FUNCTION_BLOCK FB_Alarm EXTENDS Tc3_EventLogger.FB_TcAlarm
VAR_INPUT
	stEventEntry : TcEventEntry;		// TcEventEntry to be created and send
	bSetAlarm : BOOL; // Boolean to set create alarm
	bResetAlarm : BOOL; // Boolean to reset(clear) alarm
	bWithConfirmation: BOOL; // Boolean to set alarm with confirmation
	bResetConfirmation: BOOL; // Boolean to reset alarm with confirmation
END_VAR
VAR_OUTPUT
END_VAR
VAR
	rTrigSetAlarm : R_TRIG;
	rTrigResetAlarm : R_TRIG;
END_VAR

rTrigSetAlarm(CLK:= bSetAlarm); // Using rising trigger to make sure to set alarms only once
rTrigResetAlarm(CLK:= bResetAlarm); // Using rising trigger to make sure to reset(clear) alarm only once


M_SetAlarm(bCommand:= bSetAlarm); // Calling method to set alarm
M_ResetAlarm(bCommand:= bResetAlarm); // Calling method to reset alarm

METHOD M_ResetAlarm : HRESULT
VAR_INPUT
		bCommand: BOOL;
END_VAR

VAR
END_VAR
// ======================================================================

IF bCommand THEN
	
	F_SucceededHR(Clear(0,bResetConfirmation),M_ResetAlarm); // Clearing the alarm using TC library FB_TcAlarm
	
END_IF

// ======================================================================
END_METHOD

METHOD M_SetAlarm : HRESULT
VAR_INPUT
	bCommand : BOOL;
END_VAR
// ======================================================================
// Create Alarm and Raise it 
IF bCommand THEN
	
		IF F_SucceededHr(CreateEx(stEventEntry, bWithConfirmation, 0), M_SetAlarm) THEN // Create Alaram
			F_SucceededHr(Raise(0), M_SetAlarm); // Raise Alarm
		END_IF

END_IF	
// ======================================================================
END_METHOD

END_FUNCTION_BLOCK

(* stored: Version 1.1.0.1, ProductVersion 3.1.4024.6
   POU FB_Alarm: Id {21dddc1d-62a8-4ab0-80db-5e55ed64db58}, SpecialFunc None
   Method M_ResetAlarm: Id {89791be2-556d-480b-b828-5f23c9161760}
   Method M_SetAlarm: Id {6add7e2c-d31f-46b5-90d6-e5cb1861d016} *)
